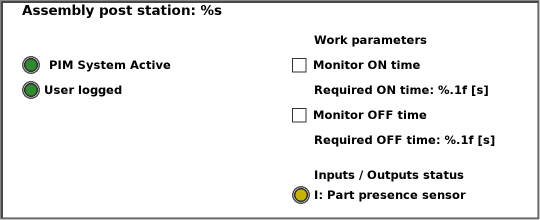
VISUALIZATION vAssemblyPost_Status  // 540x220
VAR_IN_OUT
	fbData:fbAssemblyPost;
END_VAR
    Rectangle (1,1 538x218), "Assembly post station: %s", text variable: fbData.stStationData.sNazwaStanowiska
    RoundedRectangle (18,55 193x20), "PIM System Active", colour toggle: NOT fbData.bPIM_Active
    Rectangle (311,80 200x20), "Required ON time: %.1f [s]", text variable: fbData.stWorkParams.rRequiredTimeON, input disabled if: NOT GVL.fbUserLogin.bPermissionGranted
        OnMouseClick: write the text variable via Default, min 0.5, max 30, title 'Required ON time', format %.1f
    Label (41,80 170x20), "User logged"
    Lamp1 (21,80 20x20), variable: fbData.bUserLogged, style: Lamp-Lamp1-Green
    Label (311,185 170x20), "I: Part presence sensor"
    Lamp1 (291,185 20x20), variable: fbData.fbPartFiltered.Q, style: Lamp-Lamp1-Yellow
    Label (311,165 170x20), "Inputs / Outputs status"
    Lamp1 (21,55 20x20), variable: fbData.bPIM_Active, style: Lamp-Lamp1-Green
    Rectangle (311,130 200x20), "Required OFF time: %.1f [s]", text variable: fbData.stWorkParams.rRequiredTimeOFF, input disabled if: NOT GVL.fbUserLogin.bPermissionGranted
        OnMouseClick: write the text variable via Default, min 0.5, max 30, title 'Required OFF time', format %.1f
    Checkbox (290,55 20x20), variable: fbData.stWorkParams.bMonitorON_Time, input disabled if: NOT GVL.fbUserLogin.bPermissionGranted
    Label (310,55 170x20), "Monitor ON time"
    Checkbox (290,105 20x20), variable: fbData.stWorkParams.bMonitorOFF_Time, input disabled if: NOT GVL.fbUserLogin.bPermissionGranted
    Label (310,105 170x20), "Monitor OFF time"
    Label (311,30 170x20), "Work parameters"
END_VISUALIZATION

(* stored: Version 1.1.0.1, ProductVersion 3.1.4024.12
   Visu vAssemblyPost_Status: Id {c688e117-1af3-4822-ab18-d7296b8e5bd2} *)
